FUNCTION_BLOCK GE_LINT (* IEC 61131-3,Table 28#6 *)
  (* Standard: 61131-3 *)
  (* Version 0.0, 2004-12-15, JHC, Rockwell Automation, Converted from SRC format. *)
  (* Compiler header: package fb.rt.plc.comp; *)
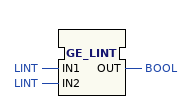
  VAR_INPUT
    IN1 : LINT;
    IN2 : LINT;
  END_VAR
  VAR_OUTPUT
    OUT : BOOL;
  END_VAR
END_FUNCTION_BLOCK
